(* IEC 61131-3 sources: MotionTestBenchMaster/Logical/30_MC/Task/Cyclic03/MC_INTERFACE (part 3) *)

(* ---- PAR_Profibus.st ---- *)
ACTION PAR_Profibus:
	MC_InputOutput.Network.Machine.Parameters.Cam02OnValue		:= UINT_TO_REAL(USINT_TO_UINT(IO_MCRaw.Input.PAR[1])	+ (USINT_TO_UINT(IO_MCRaw.Input.PAR[0])	* 16#100)) / 10.0;
	MC_InputOutput.Network.Machine.Parameters.Cam02OffValue		:= UINT_TO_REAL(USINT_TO_UINT(IO_MCRaw.Input.PAR[3])	+ (USINT_TO_UINT(IO_MCRaw.Input.PAR[2])	* 16#100)) / 10.0;
	MC_InputOutput.Network.Machine.Parameters.Cam02AdvTime		:= UINT_TO_REAL(USINT_TO_UINT(IO_MCRaw.Input.PAR[5])	+ (USINT_TO_UINT(IO_MCRaw.Input.PAR[4])	* 16#100)) / 10.0;
	MC_InputOutput.Network.Machine.Parameters.Cam02Pulse		:= IO_MCRaw.Input.PAR[6];
	IO_MCRaw.Input.PAR[7];
	IO_MCRaw.Input.PAR[8];
	IO_MCRaw.Input.PAR[9];
	MC_InputOutput.Network.Machine.Parameters.Cam03OnValue		:= UINT_TO_REAL(USINT_TO_UINT(IO_MCRaw.Input.PAR[11])	+ (USINT_TO_UINT(IO_MCRaw.Input.PAR[10])	* 16#100)) / 10.0;
	MC_InputOutput.Network.Machine.Parameters.Cam03OffValue		:= UINT_TO_REAL(USINT_TO_UINT(IO_MCRaw.Input.PAR[13])	+ (USINT_TO_UINT(IO_MCRaw.Input.PAR[12])	* 16#100)) / 10.0;
	MC_InputOutput.Network.Machine.Parameters.Cam03AdvTime		:= UINT_TO_REAL(USINT_TO_UINT(IO_MCRaw.Input.PAR[15])	+ (USINT_TO_UINT(IO_MCRaw.Input.PAR[14])	* 16#100)) / 10.0;
	MC_InputOutput.Network.Machine.Parameters.Cam03Pulse		:= IO_MCRaw.Input.PAR[16];
	IO_MCRaw.Input.PAR[17];
	IO_MCRaw.Input.PAR[18];
	IO_MCRaw.Input.PAR[19];
	MC_InputOutput.Network.Machine.Parameters.Cam04OnValue		:= UINT_TO_REAL(USINT_TO_UINT(IO_MCRaw.Input.PAR[21])	+ (USINT_TO_UINT(IO_MCRaw.Input.PAR[20])	* 16#100)) / 10.0;
	MC_InputOutput.Network.Machine.Parameters.Cam04OffValue		:= UINT_TO_REAL(USINT_TO_UINT(IO_MCRaw.Input.PAR[23])	+ (USINT_TO_UINT(IO_MCRaw.Input.PAR[22])	* 16#100)) / 10.0;
	MC_InputOutput.Network.Machine.Parameters.Cam04AdvTime		:= UINT_TO_REAL(USINT_TO_UINT(IO_MCRaw.Input.PAR[25])	+ (USINT_TO_UINT(IO_MCRaw.Input.PAR[24])	* 16#100)) / 10.0;
	MC_InputOutput.Network.Machine.Parameters.Cam04Pulse  		:= IO_MCRaw.Input.PAR[26];
	IO_MCRaw.Input.PAR[27];
	IO_MCRaw.Input.PAR[28];
	IO_MCRaw.Input.PAR[29];
	MC_InputOutput.Network.Machine.Parameters.Cam05OnValue		:= UINT_TO_REAL(USINT_TO_UINT(IO_MCRaw.Input.PAR[31])	+ (USINT_TO_UINT(IO_MCRaw.Input.PAR[30])	* 16#100)) / 10.0;
	MC_InputOutput.Network.Machine.Parameters.Cam05OffValue		:= UINT_TO_REAL(USINT_TO_UINT(IO_MCRaw.Input.PAR[33])	+ (USINT_TO_UINT(IO_MCRaw.Input.PAR[32])	* 16#100)) / 10.0;
	MC_InputOutput.Network.Machine.Parameters.Cam05AdvTime		:= UINT_TO_REAL(USINT_TO_UINT(IO_MCRaw.Input.PAR[35])	+ (USINT_TO_UINT(IO_MCRaw.Input.PAR[34])	* 16#100)) / 10.0;
	MC_InputOutput.Network.Machine.Parameters.Cam05Pulse  		:= IO_MCRaw.Input.PAR[36];
	IO_MCRaw.Input.PAR[37];
	IO_MCRaw.Input.PAR[38];
	IO_MCRaw.Input.PAR[39];
	MC_InputOutput.Network.Machine.Parameters.Cam06OnValue		:= UINT_TO_REAL(USINT_TO_UINT(IO_MCRaw.Input.PAR[41])	+ (USINT_TO_UINT(IO_MCRaw.Input.PAR[40])	* 16#100)) / 10.0;
	MC_InputOutput.Network.Machine.Parameters.Cam06OffValue		:= UINT_TO_REAL(USINT_TO_UINT(IO_MCRaw.Input.PAR[43])	+ (USINT_TO_UINT(IO_MCRaw.Input.PAR[42])	* 16#100)) / 10.0;
	MC_InputOutput.Network.Machine.Parameters.Cam06AdvTime		:= UINT_TO_REAL(USINT_TO_UINT(IO_MCRaw.Input.PAR[45])	+ (USINT_TO_UINT(IO_MCRaw.Input.PAR[44])	* 16#100)) / 10.0;
	MC_InputOutput.Network.Machine.Parameters.Cam06Pulse  		:= IO_MCRaw.Input.PAR[46];
	IO_MCRaw.Input.PAR[47];
	IO_MCRaw.Input.PAR[48];
	IO_MCRaw.Input.PAR[49];
	MC_InputOutput.Network.Machine.Parameters.Cam07OnValue		:= UINT_TO_REAL(USINT_TO_UINT(IO_MCRaw.Input.PAR[51])	+ (USINT_TO_UINT(IO_MCRaw.Input.PAR[50])	* 16#100)) / 10.0;
	MC_InputOutput.Network.Machine.Parameters.Cam07OffValue		:= UINT_TO_REAL(USINT_TO_UINT(IO_MCRaw.Input.PAR[53])	+ (USINT_TO_UINT(IO_MCRaw.Input.PAR[52])	* 16#100)) / 10.0;
	MC_InputOutput.Network.Machine.Parameters.Cam07AdvTime		:= UINT_TO_REAL(USINT_TO_UINT(IO_MCRaw.Input.PAR[55])	+ (USINT_TO_UINT(IO_MCRaw.Input.PAR[54])	* 16#100)) / 10.0;
	MC_InputOutput.Network.Machine.Parameters.Cam07Pulse  		:= IO_MCRaw.Input.PAR[56];
	IO_MCRaw.Input.PAR[57];
	IO_MCRaw.Input.PAR[58];
	IO_MCRaw.Input.PAR[59];
	MC_InputOutput.Network.Machine.Parameters.Cam08OnValue		:= UINT_TO_REAL(USINT_TO_UINT(IO_MCRaw.Input.PAR[61])	+ (USINT_TO_UINT(IO_MCRaw.Input.PAR[60])	* 16#100)) / 10.0;
	MC_InputOutput.Network.Machine.Parameters.Cam08OffValue		:= UINT_TO_REAL(USINT_TO_UINT(IO_MCRaw.Input.PAR[63])	+ (USINT_TO_UINT(IO_MCRaw.Input.PAR[62])	* 16#100)) / 10.0;
	MC_InputOutput.Network.Machine.Parameters.Cam08AdvTime		:= UINT_TO_REAL(USINT_TO_UINT(IO_MCRaw.Input.PAR[65])	+ (USINT_TO_UINT(IO_MCRaw.Input.PAR[64])	* 16#100)) / 10.0;
	MC_InputOutput.Network.Machine.Parameters.Cam08Pulse  		:= IO_MCRaw.Input.PAR[66];
	IO_MCRaw.Input.PAR[67];
	IO_MCRaw.Input.PAR[68];
	IO_MCRaw.Input.PAR[69];
	MC_InputOutput.Network.Filler.Parameters.TorqueError.In[1]	:= UINT_TO_REAL(USINT_TO_UINT(IO_MCRaw.Input.PAR[71])	+ (USINT_TO_UINT(IO_MCRaw.Input.PAR[70])	* 16#100)) / 10.0;
	MC_InputOutput.Network.Filler.Parameters.TorqueError.In[2]	:= UINT_TO_REAL(USINT_TO_UINT(IO_MCRaw.Input.PAR[73])	+ (USINT_TO_UINT(IO_MCRaw.Input.PAR[72])	* 16#100)) / 10.0;
	MC_InputOutput.Network.Filler.Parameters.TorqueError.In[3]	:= UINT_TO_REAL(USINT_TO_UINT(IO_MCRaw.Input.PAR[75])	+ (USINT_TO_UINT(IO_MCRaw.Input.PAR[74])	* 16#100)) / 10.0;
	MC_InputOutput.Network.Filler.Parameters.TorqueError.In[4]	:= UINT_TO_REAL(USINT_TO_UINT(IO_MCRaw.Input.PAR[77])	+ (USINT_TO_UINT(IO_MCRaw.Input.PAR[76])	* 16#100)) / 10.0;
	MC_InputOutput.Network.Filler.Parameters.TorqueError.In[5]	:= UINT_TO_REAL(USINT_TO_UINT(IO_MCRaw.Input.PAR[79])	+ (USINT_TO_UINT(IO_MCRaw.Input.PAR[78])	* 16#100)) / 10.0;
	MC_InputOutput.Network.Filler.Parameters.TorqueError.In[6]	:= UINT_TO_REAL(USINT_TO_UINT(IO_MCRaw.Input.PAR[81])	+ (USINT_TO_UINT(IO_MCRaw.Input.PAR[80])	* 16#100)) / 10.0;
	MC_InputOutput.Network.Filler.Parameters.TorqueError.In[7]	:= UINT_TO_REAL(USINT_TO_UINT(IO_MCRaw.Input.PAR[83])	+ (USINT_TO_UINT(IO_MCRaw.Input.PAR[82])	* 16#100)) / 10.0;
	MC_InputOutput.Network.Filler.Parameters.TorqueError.In[8]	:= UINT_TO_REAL(USINT_TO_UINT(IO_MCRaw.Input.PAR[85])	+ (USINT_TO_UINT(IO_MCRaw.Input.PAR[84])	* 16#100)) / 10.0;
	MC_InputOutput.Network.Filler.Parameters.TorqueError.In[9]	:= UINT_TO_REAL(USINT_TO_UINT(IO_MCRaw.Input.PAR[87])	+ (USINT_TO_UINT(IO_MCRaw.Input.PAR[86])	* 16#100)) / 10.0;
	MC_InputOutput.Network.Filler.Parameters.TorqueError.In[10]	:= UINT_TO_REAL(USINT_TO_UINT(IO_MCRaw.Input.PAR[89])	+ (USINT_TO_UINT(IO_MCRaw.Input.PAR[88])	* 16#100)) / 10.0;
	MC_InputOutput.Network.Filler.Parameters.TorqueError.Main	:= UINT_TO_REAL(USINT_TO_UINT(IO_MCRaw.Input.PAR[91])	+ (USINT_TO_UINT(IO_MCRaw.Input.PAR[90])	* 16#100)) / 10.0;
	MC_InputOutput.Network.Filler.Parameters.TorqueError.Out[1]	:= UINT_TO_REAL(USINT_TO_UINT(IO_MCRaw.Input.PAR[93])	+ (USINT_TO_UINT(IO_MCRaw.Input.PAR[92])	* 16#100)) / 10.0;
	MC_InputOutput.Network.Filler.Parameters.TorqueError.Out[2]	:= UINT_TO_REAL(USINT_TO_UINT(IO_MCRaw.Input.PAR[95])	+ (USINT_TO_UINT(IO_MCRaw.Input.PAR[94])	* 16#100)) / 10.0;
	MC_InputOutput.Network.Filler.Parameters.TorqueError.Out[3]	:= UINT_TO_REAL(USINT_TO_UINT(IO_MCRaw.Input.PAR[97])	+ (USINT_TO_UINT(IO_MCRaw.Input.PAR[96])	* 16#100)) / 10.0;
	MC_InputOutput.Network.Filler.Parameters.TorqueError.Out[4]	:= UINT_TO_REAL(USINT_TO_UINT(IO_MCRaw.Input.PAR[99])	+ (USINT_TO_UINT(IO_MCRaw.Input.PAR[98])	* 16#100)) / 10.0;
	MC_InputOutput.Network.Filler.Parameters.TorqueError.Out[5]	:= UINT_TO_REAL(USINT_TO_UINT(IO_MCRaw.Input.PAR[101]) + (USINT_TO_UINT(IO_MCRaw.Input.PAR[100])	* 16#100)) / 10.0;
	MC_InputOutput.Network.Filler.Parameters.TorqueError.Out[6]	:= UINT_TO_REAL(USINT_TO_UINT(IO_MCRaw.Input.PAR[103]) + (USINT_TO_UINT(IO_MCRaw.Input.PAR[102])	* 16#100)) / 10.0;
	IO_MCRaw.Input.PAR[104];
	IO_MCRaw.Input.PAR[105];
END_ACTION

(* ---- Variables.var ---- *)
VAR
	xModuleOutletInizialized : BOOL; (*1.7.2*)
	xModuleInletInizialized : BOOL; (*1.7.2*)
	xModuleFillerInizialized : BOOL; (*1.7.2*)
	uiHmiAxisIndex : UINT;
	uiAxisIndex : UINT;
	tofShiftDoneOff : TOF;
	xPhasingRunning : BOOL;
	xAxisInVelocityControl : BOOL;
	iTempInt : INT; (*v1.2*)
	iTempInt2 : INT; (*v1.2*)
END_VAR
